// TIA Portal V19 export
FUNCTION "A03_TrkManager_CALL" : Void   // FC87, LAD
// stored: SetENOAutomatically false
BEGIN

REGION Network 1
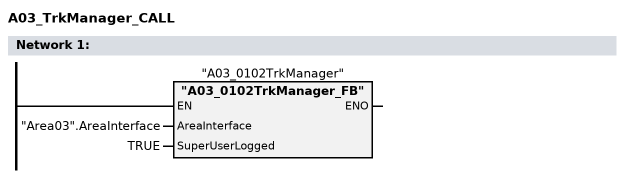
   RUNG wire#powerrail
      "A03_0102TrkManager"(AreaInterface := "Area03".AreaInterface, SuperUserLogged := TRUE)
   END_RUNG
   // the same network as SCL:
   "A03_0102TrkManager"(AreaInterface := "Area03".AreaInterface, SuperUserLogged := TRUE);   // "A03_0102TrkManager_FB"
END_REGION
END_FUNCTION
